//Test setups (fixtures), for PMPS components
PROGRAM TestSetups
VAR
	fbBPTMTest	:	FB_BPTM_Test;
	fbSafeBPCompareTest	:	FB_SafeBPCompare_Test;
	fbevWithinSpecTest	:	FB_evWithinSpec_Test;
	fbPEWTest	:	FB_PhotonEnergyWatcher_Test;
	fbFFTest	:	FB_FastFault_Test;
	fbArbiterTest	:	FB_Arbiter_Test;
END_VAR

TcUnit.RUN();

END_PROGRAM

(* stored: Version 1.1.0.1, ProductVersion 3.1.4022.18
   POU TestSetups: Id {b76e0cd1-9067-0211-3640-810a8ad26b8e}, SpecialFunc None *)
